ABB RobotStudio station: CellaRobotizzata_20210416-193104.rsstn

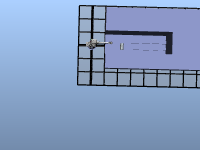
Station Solution8 (saved by RobotStudio 7.0.8504.151)
Controller IRB_4600_20kg_2.50m, task T_ROB1: task frame (RAPID world) sits at (0, 0, 900) mm in the station
Controller IRB_4600_20kg_2.50m
  mechanical unit ROB_1: IRB4600_20_250_C_01, 6 joints, base frame (0, 0, 0) mm
Layout (positions relative to the parent item):
  - IRB4600_20_250_C_01 [mechanism, from Robots\IRB4600_20_250_C_G_01.rslib] at (0, 0, 900) mm; joint values [0, 0, 0, 0, 0.5236, 0] (rad or m)
  - CentroDiLavoro [part] at (1000, 0, 1318.5) mm
  - PalletLavoro [part] at (1897.62, -173.66, 1318.5) mm
  - PalletLavoro_2 [part] at (1012.29, -173.66, 1318.5) mm
  - Basamento_robot_2 [part] at (0, 0, 900) mm
  - testata_motore [part] at (2199.69, -143.24, 1442.67) mm, rotated rx 90 ry 0 rz 0 deg
